{attribute addProperty BoxType "EL5151-0090-0016"}
{attribute addProperty Id "StatusAT %I*Status_BAC5C70E1621Counter_valueAT %I*UINT16217Latch_valueAT %I*UINT16218"}
{attribute addProperty CRC "2036154"}
{attribute addProperty SizeInBites "48"}
{attribute addProperty SizeInBytes "6"}
TYPE ENC_Status_compact_001F11BA :
STRUCT
	{attribute addProperty Name "Status"}
	Status AT %I* : Status_BAC5C70E;
	{attribute addProperty Name "Counter_value"}
	Counter_value AT %I* : UINT;
	{attribute addProperty Name "Latch_value"}
	Latch_value AT %I* : UINT;
END_STRUCT
END_TYPE

(* stored: Version 1.2.0.0, ProductVersion 3.1.4024.9
   DUT ENC_Status_compact_001F11BA: Id {874586c1-5194-4c56-becf-dd3fcf08452b} *)
